FOR i:=0 TO 7 DO
	IF ((wCrc_buff AND 16#0001) XOR (byInput AND 16#01)) = 1 THEN
		wX16 := 16#8408;
	ELSE
		wX16 := 16#0000;
	END_IF
	wCrc_buff := SHR(wCrc_buff, 1);
	wCrc_buff := wCrc_buff   XOR wX16;
	byInput := SHR (byInput, 1);
END_FOR

F_CRC_CALC := wCrc_buff;

END_FUNCTION

// ---- POUs/Various/F_ScaleLREAL.TcPOU
//==================================================================================================
//							Beckhoff Automation Poland
//									30.03.2017
//			Funkcja skalujaca
// 	v1.0	|| TC v 3.1.4020.32		|| - pierwsza wersja
//==================================================================================================
FUNCTION F_ScaleLREAL: LREAL
VAR_INPUT
	lrValue									: LREAL;				// Zmienna skalowana
	lrXmin									: LREAL;				// Dolny zakres zmiennej przeskalowanej
	lrXmax									: LREAL;				// Gorny zakres zmiennej przeskalowanej
	lrYmin									: LREAL;				// Dolny zakres zmiennej skalowanej
	lrYmax									: LREAL;				// Gorny zakres zmiennej skalowanej
	bLimits									: BOOL;					// Ogranicz wyjscie w przedziale lrYmin : lrYmax
END_VAR
VAR
	lrfA									: LREAL;				// Wspolczynnik kierunkowy prostej
	lrfB									: LREAL;				// Wspolczynnik przesuniecia prostej
END_VAR

IF (((lrXmax - lrXmin) < 0.01) AND ((lrXmax - lrXmin) > -0.01)) THEN
	F_ScaleLREAL := lrYmin;
ELSE
	lrfA := (lrYmax - lrYmin) / (lrXmax - lrXmin);
	lrfB := lrYmax - lrfA * lrXmax;
	F_ScaleLREAL := lrfA * lrValue + lrfB;
END_IF;
// LIMITY - opcja
IF bLimits THEN
	IF lrYmin < lrYmax THEN
		F_ScaleLREAL := LIMIT(lrYmin, F_ScaleLREAL, lrYmax);
	ELSE
		F_ScaleLREAL := LIMIT(lrYmax, F_ScaleLREAL, lrYmin);		
	END_IF	
END_IF

END_FUNCTION

// ---- POUs/Various/TONR.TcPOU
FUNCTION_BLOCK TONR
VAR_INPUT
	IN 			: BOOL;		// Start input
	RIN			: BOOL;		// Reset input
	PT			: TIME;		// Maximum duration of time recording
END_VAR
VAR_OUTPUT
	Q			: BOOL;		// Output tht is set when time PT expires
	ET			: TIME;		// Accumulated time
END_VAR
VAR
	startTime 	: TIME;
	inputTrig	: R_TRIG;
	resetTrig	: R_TRIG;
END_VAR

(* Update start time *)
inputTrig(CLK := IN AND NOT RIN);
startTime := SEL(inputTrig.Q, startTime, TIME() - ET); 

(* Reset timer *)
resetTrig(CLK := RIN);
ET := SEL(resetTrig.Q, ET, T#0S);

(* Set outputs *)
ET 	:= SEL(IN AND NOT RIN, ET, TIME() - startTime);
Q 	:= SEL(IN AND ET >= PT, FALSE, TRUE);

END_FUNCTION_BLOCK
